TEXTLIST StationAckMode_txt
  0 = 'Time'
  1 = 'External Ack'
   = ''
END_TEXTLIST

(* stored: Version 1.1.0.1, ProductVersion 3.1.4024.11
   TextList StationAckMode_txt: Id {08c45bd7-6689-43d8-b9c6-fa89f3cc89ea} *)
